(*

.. <legal notes>

legal notes
=================
| SPDX-FileCopyrightText: © 2026 Oleksandr Tiutyk <trofimich@gmail.com>
| SPDX-License-Identifier: LGPL-3.0-only
| For details check: LGPL-3.0-only_

.. _LGPL-3.0-only: https://www.gnu.org/licenses/lgpl-3.0.en.html

.. </legal notes>

*)

INTERFACE IAutomationRunner EXTENDS Core.IObject

{attribute 'monitoring' := 'call'}
PROPERTY FINAL CodeExecutionPhase : BOOL
GET
END_GET
END_PROPERTY

{attribute 'monitoring' := 'call'}
PROPERTY FINAL CycleCounter : LWORD
GET
END_GET
END_PROPERTY

METHOD FINAL Execute
VAR_IN_OUT CONSTANT
	controllers : ARRAY [*] OF IAutomationController;
END_VAR
END_METHOD

{attribute 'monitoring' := 'call'}
PROPERTY FINAL State : AUTOMATION_RUNNER_STATE
GET
END_GET
END_PROPERTY

{attribute 'monitoring' := 'call'}
PROPERTY StateName : STRING
GET
END_GET
END_PROPERTY

END_INTERFACE

(* stored: Version 1.1.0.1
   Itf IAutomationRunner: Id {276b0ed1-ca71-445c-ba80-324e25054832}
   Property CodeExecutionPhase: Id {87d579d2-6769-4f81-b459-0ad410ea60da}
   Get Get: Id {eed90592-18ca-4fae-ba5d-68502892d691}
   Property CycleCounter: Id {2afeb81b-86ed-40c7-b2f1-2294697c62ef}
   Get Get: Id {1107fa50-7f06-4d4e-9e15-119390b0c3e5}
   Method Execute: Id {77862fb4-f337-4ebd-a567-9b8cb57e2f0a}
   Property State: Id {08c8944f-e3b7-41a3-9ea3-12dd40206d8d}
   Get Get: Id {71fcea67-0c10-4775-921c-1b22e59917c9}
   Property StateName: Id {bc56f41a-11b5-42f2-9300-61a1f839f72b}
   Get Get: Id {9fbb0b29-ff34-40eb-a365-b63072d06173} *)
